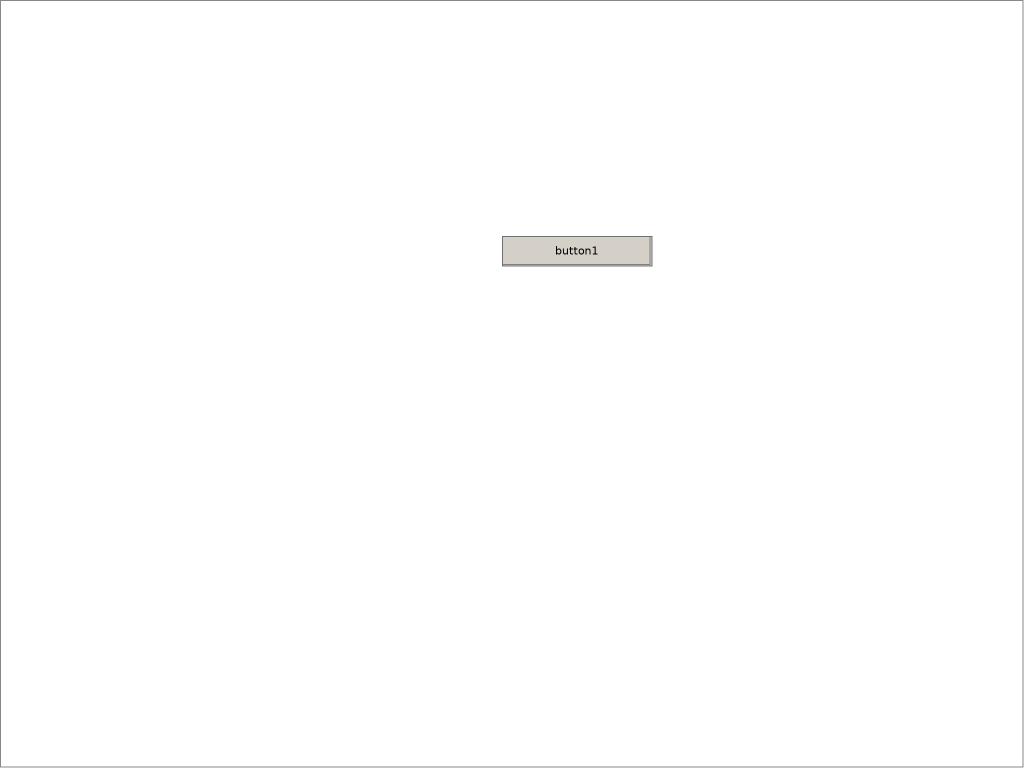
VISUALIZATION visu_a10  // 1024x768
    Button (502,236 150x30), "button1"
END_VISUALIZATION

(* stored: Version 1.1.0.1, ProductVersion 3.1.4024.12
   Visu visu_a10: Id {81ad7c19-6766-40ab-9d0e-11804f283e42} *)
